{attribute 'qualified_only'}
{attribute 'strict'}
TYPE ENUM_CoolingMethod :
(
	fdc := 0,
	laminair := 1
);
END_TYPE

(* stored: Version 1.1.0.1, ProductVersion 3.1.4024.2
   DUT ENUM_CoolingMethod: Id {b49117a2-f3a6-4981-a4a3-5220bd6d9f5a} *)
